TYPE ST_PumpCommand :
STRUCT
	bRunBySpeed  : BOOL;
    bRunByVolume : BOOL;
    bStop        : BOOL;
    bActive      : BOOL;
    eDirection   : E_PumpDirection;
    rSpeed       : REAL; // % or RPM
    rVolume      : REAL; // mL or user unit
	iDistance	 : UINT; // Revs number
    bBusy        : BOOL;
END_STRUCT
END_TYPE

(* stored: Version 1.1.0.1, ProductVersion 3.1.4024.12
   DUT ST_PumpCommand: Id {5f240ab5-e15e-4283-81db-9512cd15a1c1} *)
